{attribute 'linkalways'} 
{attribute 'no_explicit_call' := 'This FB is a CLASS and must be accessed using methods or properties'}
{attribute 'enable_dynamic_creation'}
FUNCTION_BLOCK _WORD EXTENDS NumericDatatypeBase
VAR
	localData : WORD;
	activeData : REFERENCE TO WORD REF= localData;
END_VAR

PROPERTY PUBLIC Address : PVOID
GET
Address := ADR(activeData);
END_GET
END_PROPERTY

METHOD PUBLIC ClearReference
VAR_INPUT
END_VAR
activeData REF= localData;
END_METHOD

METHOD PUBLIC Clone : I_Datatype
VAR
    pClone : POINTER TO _WORD;
END_VAR
pClone := __NEW(_WORD(InitialValue := Value));
Clone := pClone^;
END_METHOD

METHOD FB_init : BOOL
VAR_INPUT
	bInitRetains : BOOL; // if TRUE, the retain variables are initialized (warm start / cold start)
	bInCopyCode : BOOL;  // if TRUE, the instance afterwards gets moved WORDo the copy code (online change)
	InitialValue : WORD;
END_VAR
localData := InitialValue;
END_METHOD

PROPERTY PUBLIC IsFloat : BOOL
GET
IsFloat := FALSE;
END_GET
END_PROPERTY

PROPERTY PUBLIC IsSigned : BOOL
GET
IsSigned := FALSE;
END_GET
END_PROPERTY

PROPERTY PUBLIC LowerBound : WORD
GET
LowerBound := DatatypeLimits.WORD_LOWER_LIMIT;
END_GET
END_PROPERTY

METHOD PUBLIC MakeReferenceTo
VAR_INPUT
	ReferenceTarget : REFERENCE TO WORD;
END_VAR
activeData REF= ReferenceTarget;
END_METHOD

METHOD PROTECTED SerializeLowerbound
VAR_INPUT
	Serializer : I_Serializer;
END_VAR
Serializer.AddWord(Lowerbound);
END_METHOD

METHOD PROTECTED SerializeUpperbound
VAR_INPUT
	Serializer : I_Serializer;
END_VAR
Serializer.AddWord(Upperbound);
END_METHOD

METHOD PUBLIC SerializeWith
VAR_INPUT
	Serializer : I_Serializer;
END_VAR
Serializer.AddWord(activeData);
END_METHOD

PROPERTY PUBLIC Size : UDINT
GET
Size := SIZEOF(activeData);
END_GET
END_PROPERTY

METHOD TryDeserializeFrom : BOOL
VAR_INPUT
	Deserializer : I_Deserializer;
	Feedback : I_DeserializerFeedback;
END_VAR
TryDeserializeFrom := Deserializer.TryGetWord(activeData, Feedback);
END_METHOD

METHOD TryMakeReferenceTo : BOOL
VAR_INPUT
	Target : I_Datatype;
END_VAR
VAR
	pTargetData : POINTER TO WORD;
END_VAR
IF NOT (Target.TypeName = TypeName) THEN
	RETURN;
END_IF

pTargetData := Target.Address;
activeData REF= pTargetData^;
TryMakeReferenceTo := TRUE;
END_METHOD

PROPERTY PUBLIC TypeName : T_MAXSTRING
GET
TypeName := 'WORD';
END_GET
END_PROPERTY

PROPERTY PUBLIC UpperBound : WORD
GET
UpperBound :=  DatatypeLimits.WORD_UPPER_LIMIT;
END_GET
END_PROPERTY

PROPERTY PUBLIC Value : WORD
GET
Value := activeData;
END_GET
SET
activeData := Value;
END_SET
END_PROPERTY

END_FUNCTION_BLOCK

(* stored: Version 1.1.0.1, ProductVersion 3.1.4024.12
   POU _WORD: Id {3a58d2d7-f996-08b8-388d-4e702b3985a4}, SpecialFunc None
   Folder Constructor: Id {69cad55d-99cd-01a6-044c-574b9b1a9e94}
   Folder Protected: Id {e43fcdb7-e8a4-0d23-079c-925b27974933}
   Property Address: Id {9feaacf0-5d7c-0919-232b-c699e8c20f96}
   Get Get: Id {57808a81-6e08-0bb1-3d6b-b79212e235d9}
   Method ClearReference: Id {42685fd8-f653-0ffd-1d21-00a6bcff3f2f}
   Method Clone: Id {78db9abe-2b4c-0ebf-2ad5-ffac12f515e5}
   Method FB_init: Id {67c81700-b958-0ba1-3712-498a07586577}
   Property IsFloat: Id {d2325832-e81a-08a0-164b-27f57ae76f8a}
   Get Get: Id {31931ff9-2161-0e30-3887-995ad9406e11}
   Property IsSigned: Id {37e85d4a-5b96-0d0d-027d-8c9387b026f7}
   Get Get: Id {09d7392f-d988-01e2-0e4a-73e7de92cde9}
   Property LowerBound: Id {75db9cf0-027a-0a07-1d66-6b49e137442b}
   Get Get: Id {3a88e9f5-83de-07ad-27b1-1dfd4705cbb2}
   Method MakeReferenceTo: Id {0e8b1b01-c520-01c1-3d12-49fac3a194f8}
   Method SerializeLowerbound: Id {dc6d2d22-4d4a-0139-1abb-84bbcdccbec4}
   Method SerializeUpperbound: Id {2ef5ea3e-767d-0af1-372c-36627e37d719}
   Method SerializeWith: Id {bd002f7c-1b5e-079b-284d-27e658dfa1e6}
   Property Size: Id {69de8cb6-52a3-060d-09d4-0fc7023b3b88}
   Get Get: Id {fb5f0d90-0574-03a6-2ee2-e16199452464}
   Method TryDeserializeFrom: Id {42f3a697-1247-09bc-1b43-ce4db0446be1}
   Method TryMakeReferenceTo: Id {ea593cfa-844a-0c2f-2780-d1f779c0c514}
   Property TypeName: Id {a86480b9-b762-0f4a-2cdb-6658c7e94a7e}
   Get Get: Id {fb945d17-8e78-055c-1428-68e021a3389f}
   Property UpperBound: Id {9d1ba09d-6980-0165-053b-cf805dbf9948}
   Get Get: Id {6afedcf9-4217-09c3-2aff-5a2318b4d40a}
   Property Value: Id {a4285812-b4a2-051a-1c42-e74569cabbe2}
   Get Get: Id {046c3d8f-9f11-0260-281c-17a851f14164}
   Set Set: Id {d745b444-68c8-04f8-25fd-793f711f7a59} *)
